{attribute 'qualified_only'}
VAR_GLOBAL
	Teller		:	INT;
END_VAR

(* stored: Version 1.1.0.1, ProductVersion 3.1.4024.11
   GVL GVLtest2: Id {cc2aaaaf-ace0-403f-a3ad-53ec0eb108fe} *)
